// TIA Portal V20 export
FUNCTION_BLOCK "FB_OPC_PartStatus"   // FB47, SCL
{ S7_Optimized_Access := 'TRUE' }
// stored: MemoryReserve 100, SetENOAutomatically false
   VAR_INPUT
      iGood { ExternalAccessible := 'False'; ExternalVisible := 'False'; ExternalWritable := 'False'} : Bool;
      iUnknown { ExternalAccessible := 'False'; ExternalVisible := 'False'; ExternalWritable := 'False'} : Bool;
      iBad { ExternalAccessible := 'False'; ExternalVisible := 'False'; ExternalWritable := 'False'} : Bool;
      iAbsent { ExternalAccessible := 'False'; ExternalVisible := 'False'; ExternalWritable := 'False'} : Bool;
      iPresentUnexpected { ExternalAccessible := 'False'; ExternalVisible := 'False'; ExternalWritable := 'False'} : Bool;
      iAbsentUnexpected { ExternalAccessible := 'False'; ExternalVisible := 'False'; ExternalWritable := 'False'} : Bool;
   END_VAR
   VAR_OUTPUT
      oStatus { ExternalAccessible := 'False'; ExternalVisible := 'False'; ExternalWritable := 'False'} : Byte;
   END_VAR
   VAR CONSTANT
      GOOD : Byte := 3;
      UNKNOW : Byte := 1;
      BAD : Byte := 2;
      ABSENT : Byte := 0;
      PRESENT_UNEXPECTED : Byte := 4;
      ABSENT_UNEXPECTED : Byte := 5;
      UNKNOW_STATUS : Byte := 99;
   END_VAR
BEGIN
   REGION Description header 
       //==================================================================================
       // POSALUX Swiss SA / (C) Copyright 2024
       //----------------------------------------------------------------------------------
       // Title: 
       // Comment/Function: 
       //
       // Author: Fabien WALDT
       // Engineering: TIA Portal v20
       //----------------------------------------------------------------------------------
       // Change log table:
       // Version  | Date     | Expert in charge | Changes applied
       // ---------|----------|------------------|------------------------------------
       // 00.00.01 | 20251024 | WFA              | First released version
       // ==================================================================================
   END_REGION

   REGION Status
       IF #iGood THEN
           #oStatus := #GOOD;
       ELSIF #iUnknown THEN
           #oStatus := #UNKNOW;
       ELSIF #iBad THEN
           #oStatus := #BAD;
       ELSIF #iAbsent THEN
           #oStatus := #ABSENT;
       ELSIF #iPresentUnexpected THEN
           #oStatus := #PRESENT_UNEXPECTED;
       ELSIF #iAbsentUnexpected THEN
           #oStatus := #ABSENT_UNEXPECTED;
       ELSE
           #oStatus := #UNKNOW_STATUS;
       END_IF;
   END_REGION
END_FUNCTION_BLOCK
